{attribute 'qualified_only'}
// DO NOT SET ANY OF THE CAP PARAMETERS TO 0 OR LARGER THAN MAX DINT!!!
VAR_GLOBAL CONSTANT
	DEBUGMSG_CAP	: UDINT(1..16#7FFFFFFF) := 10; // Max number of debug messages.
	DEBUGSTR_CAP	: UDINT(1..16#7FFFFFFF) := 500; // Max number of debug strings.
	
	SIGNAL_CAP		: UDINT(1..16#7FFFFFFF) := 20; // Max number of signals.
	RECEIVER_CAP	: UDINT(1..16#7FFFFFFF) := 100; // Max number of signal-receiver pairings.
END_VAR

(* stored: Version 1.1.0.1
   GVL Param: Id {bc9b684f-96ba-4011-afc3-650f65d44b69}, ParameterList True *)
